// TIA Portal V17 export
// export: Created 2024-08-07T21:43:53.0861584Z, ExportSetting WithDefaults, DisplayName Totally Integrated Automation Portal, DisplayVersion V17 Update 7, DisplayName TIA Portal Openness, DisplayVersion V17 Update 7, DisplayName TIA Portal Version Control Interface, DisplayVersion V17, DisplayName SINAMICS Startdrive Advanced, DisplayVersion V17 SP2, DisplayName SINAMICS Startdrive G110M, G120, G120C, G120D, G120P, G115D, DisplayVersion V17 SP2, DisplayName SINAMICS Startdrive G130, G150, S120, S150, SINAMICS MV, S210, DisplayVersion V17 SP2, DisplayName STEP 7 Professional, DisplayVersion V17 Update 7, DisplayName STEP 7 Safety, DisplayVersion V17 Update 6, DisplayName WinCC Advanced / Unified PC, DisplayVersion V17 Update 7
FUNCTION_BLOCK "SlidesMain"   // FB25, LAD
{ S7_Optimized_Access := 'TRUE' }
VERSION : 0.1
// stored: AutoNumber true, IsIECCheckEnabled false, IsRetainMemResEnabled false, MemoryReserve 100, SetENOAutomatically false, UDAEnableTagReadback false
   VAR
      R_TRIG_Instance { S7_SetPoint := 'True'} : R_TRIG;
      IEC_Timer_0_Instance { S7_SetPoint := 'True'} : TON_TIME;
      IEC_Timer_0_Instance_1 { S7_SetPoint := 'True'} : TOF_TIME;
      IEC_Timer_0_Instance_3 { S7_SetPoint := 'True'} : TON_TIME;
      IEC_Timer_0_Instance_5 { S7_SetPoint := 'True'} : TON_TIME;
   END_VAR
BEGIN

REGION Network 1 (SCL): NOK box from part holders
   //Check amount of parts in stock
   IF "PartHolderData".NOKBoxAmount >= "StationParameters".NOKBoxSize THEN
       "PartHolderData".NOKBoxFull := true;
   ELSE
       "PartHolderData".NOKBoxFull := FALSE;
   END_IF;

   //NOK Box signal with delay
   #R_TRIG_Instance(CLK:=NOT "iNokPartOpticalSensor");
   IF #R_TRIG_Instance.Q THEN
       "PartHolderData".NOKBoxActivated := true;
   END_IF;
   #IEC_Timer_0_Instance(IN:="PartHolderData".NOKBoxActivated,
                         PT:=t#2s);
   IF #IEC_Timer_0_Instance.Q THEN
       "PartHolderData".NOKBoxActivated := false;
   END_IF;

   //Box presence with delay
   #IEC_Timer_0_Instance_1(IN:="iNokBoxPresent",
                           PT:=t#1s,
                           Q=>"PartHolderData".NOKBoxPesent);

   //Error NOK box signal sensor
   #IEC_Timer_0_Instance_3(IN:=NOT "iNokPartOpticalSensor",
                           PT:=t#3s);
   IF #IEC_Timer_0_Instance_3.Q AND "PartHolderData".NOKBoxPesent THEN
       "SetAlarm"(AlarmNumber := 42,
                  Cell := 1,
                  Station := 99);
       ;
   END_IF;

   #IEC_Timer_0_Instance_5(IN:=NOT "iNokBoxPresent",
                           PT:=t#3s);
   IF #IEC_Timer_0_Instance_5.Q THEN
       "SetAlarm"(AlarmNumber := 40,
                  Cell := 1,
                  Station := 99);
       ;
   END_IF;

   IF "PartHolderData".NOKBoxFull THEN
       "SetAlarm"(AlarmNumber := 43,
                  Cell := 1,
                  Station := 99);
   END_IF;

   //Reset holders amounts
   "PartHolderData".ConfirmEmptyNOKBox := "PartHolderData".NOKBoxFull;
   IF "PartHolderData".EmptyNOKBoxConfirmed THEN
       "PartHolderData".NOKBoxAmount := 0;
   END_IF;
   "PartHolderData".EmptyNOKBoxConfirmed := false;
END_REGION
END_FUNCTION_BLOCK
